ABB RobotStudio station: pyramid material handling.rsstn

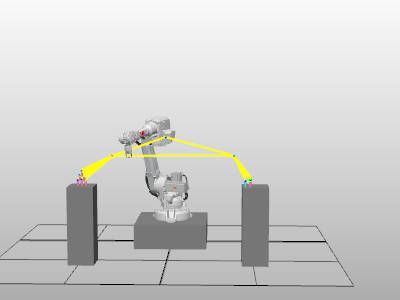
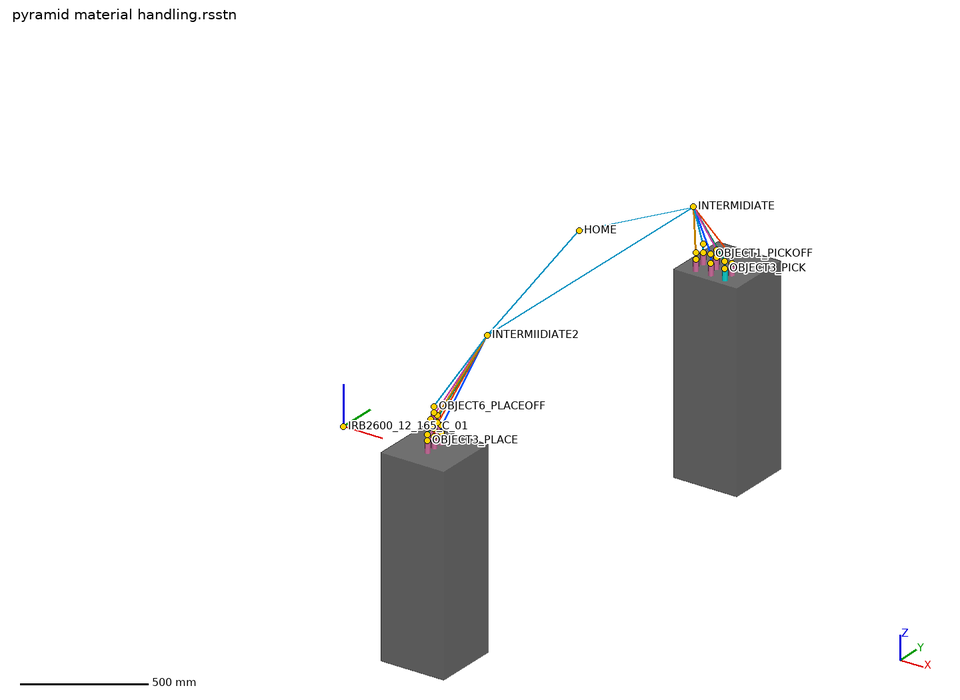
[picture v1: parts stored in the station drawn from their meshes, with robot base, taught points and paths (robot models come from the ABB library and are not in the file)]
Station Station (saved by RobotStudio 22.3.10141.1)
Controller Controller22, task T_ROB1: task frame (RAPID world) sits at (0, 0, 300) mm in the station
Controller Controller22
  mechanical unit ROB_1: IRB2600_12_165_C_01, 6 joints, base frame (0, 0, 0) mm
Layout (positions relative to the parent item):
  - concrete [part, from Libraries\concrete.rslib] at (-450, -450, 0) mm
  - IRB2600_12_165_C_01 [mechanism, from %ABB.RobotStudio.Models.IRB2600%\IRB2600_12_165_C_01.rslib] at (0, 0, 300) mm; joint values [-0.383, 0.3414, -0.2454, 0.1215, 1.4907, -1.8238] (rad or m)
  - SmartComponent_1 [smart component] at (1103.4, -433.44, 1358.47) mm, rotated rx -179.18 ry 6.95 rz -98.01 deg
      signals: DI attach
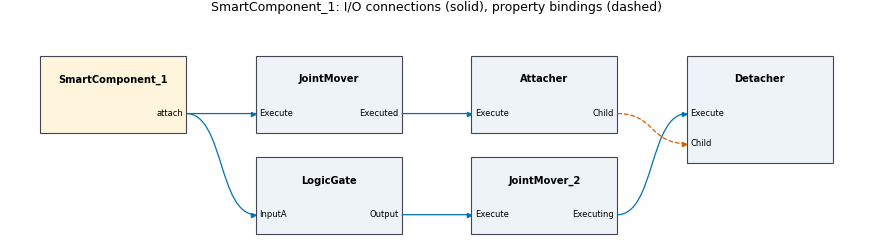
      connections:
        SmartComponent_1.attach -> JointMover.Execute
        JointMover.Executed -> Attacher.Execute
        SmartComponent_1.attach -> LogicGate.InputA
        LogicGate.Output -> JointMover_2.Execute
        JointMover_2.Executing -> Detacher.Execute
        Attacher.Child => Detacher.Child
    - Smart_Gripper_Servo_Fingers [mechanism, from Tools\ABB_Smart_Gripper_Servo_Fingers.rslib] at (0, 0, 0) mm; joint values [0.025] (rad or m)
    - JointMover [smart component, from Components\JointMover.rslib]
        properties: Mechanism=Smart_Gripper_Servo_Fingers; Relative=false; Duration=1; J1=0.023
    - JointMover_2 [smart component, from Components\JointMover.rslib]
        properties: Mechanism=Smart_Gripper_Servo_Fingers; Relative=false; Duration=1; J1=0.025
    - Attacher [smart component, from Components\Attacher.rslib]
        properties: Parent=Smart_Gripper_Servo_Fingers; Flange=0; Child=object_2; Mount=true; Offset=[0 0 0]; Orientation=[0 0 0]
    - LogicGate [smart component, from Components\LogicGate.rslib]
        properties: Operator=NOT; Delay=0
    - Detacher [smart component, from Components\Detacher.rslib]
        properties: Child=object_2; KeepPosition=true
  - table_1 [part] at (955.3, 870.39, 0) mm, size 300 x 300 x 900 mm
  - table_2 [part] at (955.3, -1114.68, 0) mm, size 300 x 300 x 900 mm
  - object [part] at (1175.36, 905.1, 900) mm, size 24 x 23.9 x 50 mm
  - object_2 [part] at (1105.3, 910.78, 900) mm, size 24 x 23.9 x 50 mm
  - object_3 [part] at (1035.28, 908.05, 900) mm, size 24 x 23.9 x 50 mm
  - object_4 [part] at (1171.86, 957.54, 900) mm, size 24 x 23.9 x 50 mm
  - object_5 [part] at (1089.6, 967.64, 900) mm, size 24 x 23.9 x 50 mm
  - object_6 [part] at (1025.27, 972.61, 900) mm, size 24 x 23.9 x 50 mm
  - object_7 [part] at (1105.3, -918.27, 900) mm, size 24 x 23.9 x 50 mm
  - object_8 [part] at (1105.3, -987.65, 951.01) mm, size 24 x 23.9 x 50 mm
  - object_9 [part] at (1105.3, -963.96, 900) mm, size 24 x 23.9 x 50 mm
  - object_10 [part] at (1105.3, -1009.85, 900) mm, size 24 x 23.9 x 50 mm
  - object_11 [part] at (1101.97, -962.11, 1002.3) mm, size 24 x 23.9 x 50 mm
  - object_12 [part] at (1104, -939.48, 950.56) mm, size 24 x 23.9 x 50 mm
Attachment: SmartComponent_1 is attached to IRB2600_12_165_C_01 / Link6
Station logic (signal -> signal, property => property):
  Controller22.attach -> SmartComponent_1.attach
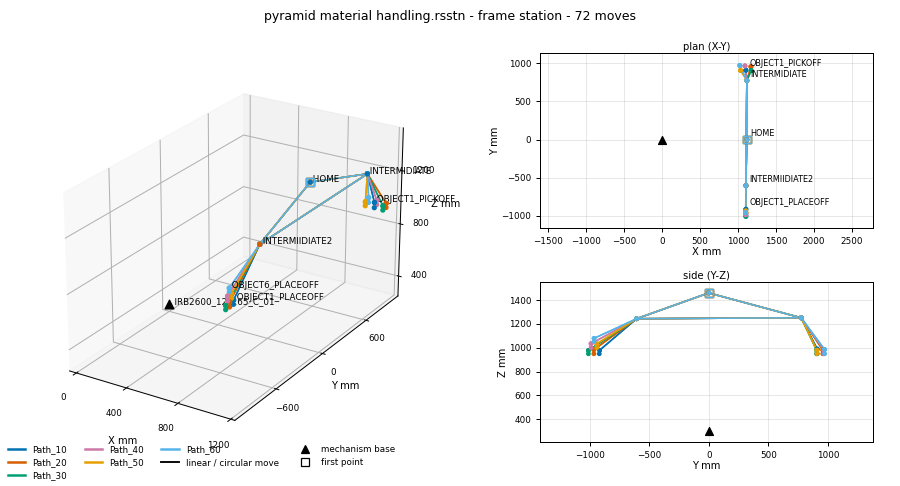
[picture p0: tool path of pyramid material handling.rsstn in frame station, 72 of 72 moves have a stored position in this frame; points joined in program order, loops and branches not executed]
Targets, tools, work objects and paths stored in the station, written as RAPID:
! task T_ROB1
MODULE CalibData
  PERS tooldata Servo:=[TRUE,[[0,0,114.2],[1,0,0,0]],[0.215,[8.7,12.3,49.2],[1,0,0,0],0.00021,0.00024,0.00009]];
ENDMODULE

! task T_ROB1
MODULE Module1
  CONST robtarget HOME:=[[1117.512260434,0,1160.4],[0.5,0,0.866025404,0],[-1,0,-1,0],[9E+09,9E+09,9E+09,9E+09,9E+09,9E+09]];
  CONST robtarget INTERMIDIATE:=[[1117.511971759,775.742463489,951.918308096],[0.499999999,-0.000000019,0.866025404,-0.000000013],[0,-1,0,0],[9E+09,9E+09,9E+09,9E+09,9E+09,9E+09]];
  CONST robtarget OBJECT1_PICK:=[[1105.303025435,910.780920196,650.000496725],[0.031021397,0.726247096,-0.685674321,-0.038125503],[0,0,-1,0],[9E+09,9E+09,9E+09,9E+09,9E+09,9E+09]];
  CONST robtarget OBJECT1_PICKOFF:=[[1105.303029888,910.780922429,689.758722238],[0.031021402,0.726247091,-0.685674327,-0.038125501],[0,0,-1,0],[9E+09,9E+09,9E+09,9E+09,9E+09,9E+09]];
  CONST robtarget INTERMIIDIATE2:=[[1105.30303417,-605.615476166,944.068794255],[0.031021378,0.726247007,-0.685674414,-0.038125531],[-1,-1,-2,0],[9E+09,9E+09,9E+09,9E+09,9E+09,9E+09]];
  CONST robtarget OBJECT1_PLACEOFF:=[[1105.303024526,-915.788819642,679.371711603],[0.031021384,0.726246988,-0.685674432,-0.038125586],[-1,-1,-2,0],[9E+09,9E+09,9E+09,9E+09,9E+09,9E+09]];
  CONST robtarget OBJECT1_PLACE:=[[1105.303040834,-918.273374791,650.000557068],[0.048952776,0.997947113,0.041056953,-0.004417227],[-1,-1,-3,0],[9E+09,9E+09,9E+09,9E+09,9E+09,9E+09]];
  CONST robtarget OBJECT2_PICKOFF:=[[1171.854966869,957.544914108,680.827668552],[0.048952841,0.997947109,0.041056966,-0.004417275],[0,-1,2,0],[9E+09,9E+09,9E+09,9E+09,9E+09,9E+09]];
  CONST robtarget OBJECT2_PICK:=[[1171.854963575,957.544912565,650.000541945],[0.048952828,0.997947111,0.041056939,-0.004417259],[0,-1,2,0],[9E+09,9E+09,9E+09,9E+09,9E+09,9E+09]];
  CONST robtarget OBJECT2_PLACE:=[[1105.303062744,-963.963465372,650.000529902],[0.032980269,-0.000000014,0.999456003,-0.000000058],[-1,0,-1,0],[9E+09,9E+09,9E+09,9E+09,9E+09,9E+09]];
  CONST robtarget OBJECT2_PLACEOFF:=[[1105.303062826,-963.963348224,684.023309799],[0.032980254,-0.000000025,0.999456003,-0.000000041],[-1,0,-1,0],[9E+09,9E+09,9E+09,9E+09,9E+09,9E+09]];
  CONST robtarget OBJECT3_PICK:=[[1175.361028607,905.095684377,650.00036776],[0.032980272,-0.000000022,0.999456003,0.000000007],[0,-1,0,0],[9E+09,9E+09,9E+09,9E+09,9E+09,9E+09]];
  CONST robtarget OBJECT3_PICKOFF:=[[1175.361033546,905.095684913,680.920223597],[0.032980305,-0.000000024,0.999456002,0.000000024],[0,-1,0,0],[9E+09,9E+09,9E+09,9E+09,9E+09,9E+09]];
  CONST robtarget OBJECT3_PLACE:=[[1105.303017361,-1009.850990253,650.000518886],[0.012165324,-0.000000073,0.999926,0.00000009],[-1,0,-1,0],[9E+09,9E+09,9E+09,9E+09,9E+09,9E+09]];
  CONST robtarget OBJECT3_PLACEOFF:=[[1105.303018098,-1009.850992621,677.758682693],[0.012165313,-0.000000049,0.999926,0.000000096],[-1,0,-1,0],[9E+09,9E+09,9E+09,9E+09,9E+09,9E+09]];
  CONST robtarget OBJECT4_PICK:=[[1092.960961058,967.413179097,650.000592066],[0.012159249,-0.00038074,0.999436296,-0.031290549],[0,-1,0,0],[9E+09,9E+09,9E+09,9E+09,9E+09,9E+09]];
  CONST robtarget OBJECT4_PICKOFF:=[[1092.960942706,967.413161677,681.87987598],[0.012159227,-0.000380743,0.999436295,-0.031290571],[0,-1,0,0],[9E+09,9E+09,9E+09,9E+09,9E+09,9E+09]];
  CONST robtarget OBJECT4_PLACE:=[[1105.303059247,-987.652451485,701.005559379],[0.01215924,-0.000380764,0.999436295,-0.03129058],[-1,-1,-1,0],[9E+09,9E+09,9E+09,9E+09,9E+09,9E+09]];
  CONST robtarget OBJECT4_PLACEOFF:=[[1105.303051029,-987.65244336,734.548047629],[0.01215925,-0.000380769,0.999436295,-0.031290587],[-1,-1,-1,0],[9E+09,9E+09,9E+09,9E+09,9E+09,9E+09]];
  CONST robtarget OBJECT5_PICK:=[[1035.27796955,908.054796965,650.000524579],[0.012159264,-0.000380741,0.999436295,-0.031290572],[0,-1,0,0],[9E+09,9E+09,9E+09,9E+09,9E+09,9E+09]];
  CONST robtarget OBJECT5_PICKOFF:=[[1035.277973445,908.054801244,679.543184231],[0.012159231,-0.000380712,0.999436294,-0.031290599],[0,-1,0,0],[9E+09,9E+09,9E+09,9E+09,9E+09,9E+09]];
  CONST robtarget OBJECT6_PICK:=[[1025.27201636,972.608074292,650.00053276],[0.012159217,-0.000380717,0.999436295,-0.031290601],[0,-1,0,0],[9E+09,9E+09,9E+09,9E+09,9E+09,9E+09]];
  CONST robtarget OBJECT6_PICKOFF:=[[1025.272009872,972.608069219,685.945409595],[0.012159225,-0.000380706,0.999436295,-0.031290591],[0,-1,0,0],[9E+09,9E+09,9E+09,9E+09,9E+09,9E+09]];
  CONST robtarget OBJECT5_PLACE:=[[1104.003999984,-939.476367792,700.564025373],[0.036344455,-0.000000046,0.999339322,0.000000022],[-1,0,-1,0],[9E+09,9E+09,9E+09,9E+09,9E+09,9E+09]];
  CONST robtarget OBJECT5_PLACEOFF:=[[1104.004008474,-939.47637643,733.669576361],[0.036344447,-0.000000033,0.999339322,0.000000026],[-1,0,-1,0],[9E+09,9E+09,9E+09,9E+09,9E+09,9E+09]];
  CONST robtarget OBJECT6_PLACE:=[[1101.97104085,-962.10978134,752.298904228],[0.036344493,0.000000006,0.999339321,0.000000002],[-1,0,-1,0],[9E+09,9E+09,9E+09,9E+09,9E+09,9E+09]];
  CONST robtarget OBJECT6_PLACEOFF:=[[1101.971036878,-962.109777758,779.422905783],[0.036344506,-0.000000004,0.99933932,-0.00000001],[-1,0,-1,0],[9E+09,9E+09,9E+09,9E+09,9E+09,9E+09]];
  PROC main()
  ENDPROC
  PROC Path_10()
    MoveL HOME,v1000,z100,Servo\WObj:=wobj0;
    MoveL INTERMIDIATE,v1000,z100,Servo\WObj:=wobj0;
    MoveL OBJECT1_PICKOFF,v1000,z100,Servo\WObj:=wobj0;
    MoveL OBJECT1_PICK,v1000,z100,Servo\WObj:=wobj0;
    WaitTime 1;
    SetDO attach,1;
    WaitTime 1;
    MoveL OBJECT1_PICKOFF,v1000,z100,Servo\WObj:=wobj0;
    MoveL INTERMIDIATE,v1000,z100,Servo\WObj:=wobj0;
    MoveL INTERMIIDIATE2,v1000,z100,Servo\WObj:=wobj0;
    MoveL OBJECT1_PLACEOFF,v1000,z100,Servo\WObj:=wobj0;
    MoveL OBJECT1_PLACE,v1000,z100,Servo\WObj:=wobj0;
    WaitTime 1;
    SetDO attach,0;
    WaitTime 1;
    MoveL OBJECT1_PLACEOFF,v1000,z100,Servo\WObj:=wobj0;
    MoveL INTERMIIDIATE2,v1000,z100,Servo\WObj:=wobj0;
    MoveL HOME,v1000,z100,Servo\WObj:=wobj0;
  ENDPROC
  PROC Path_20()
    MoveL HOME,v1000,z100,Servo\WObj:=wobj0;
    MoveL INTERMIDIATE,v1000,z100,Servo\WObj:=wobj0;
    MoveL OBJECT2_PICKOFF,v1000,z100,Servo\WObj:=wobj0;
    MoveL OBJECT2_PICK,v1000,z100,Servo\WObj:=wobj0;
    WaitTime 1;
    SetDO attach,1;
    WaitTime 1;
    MoveL OBJECT2_PICKOFF,v1000,z100,Servo\WObj:=wobj0;
    MoveL INTERMIDIATE,v1000,z100,Servo\WObj:=wobj0;
    MoveL INTERMIIDIATE2,v1000,z100,Servo\WObj:=wobj0;
    MoveL OBJECT2_PLACEOFF,v1000,z100,Servo\WObj:=wobj0;
    MoveL OBJECT2_PLACE,v1000,z100,Servo\WObj:=wobj0;
    WaitTime 1;
    SetDO attach,0;
    WaitTime 1;
    MoveL OBJECT2_PLACEOFF,v1000,z100,Servo\WObj:=wobj0;
    MoveL INTERMIIDIATE2,v1000,z100,Servo\WObj:=wobj0;
    MoveL HOME,v1000,z100,Servo\WObj:=wobj0;
  ENDPROC
  PROC Path_30()
    MoveL HOME,v1000,z100,Servo\WObj:=wobj0;
    MoveL INTERMIDIATE,v1000,z100,Servo\WObj:=wobj0;
    MoveL OBJECT3_PICKOFF,v1000,z100,Servo\WObj:=wobj0;
    MoveL OBJECT3_PICK,v1000,z100,Servo\WObj:=wobj0;
    WaitTime 1;
    SetDO attach,1;
    WaitTime 1;
    MoveL OBJECT3_PICKOFF,v1000,z100,Servo\WObj:=wobj0;
    MoveL INTERMIDIATE,v1000,z100,Servo\WObj:=wobj0;
    MoveL INTERMIIDIATE2,v1000,z100,Servo\WObj:=wobj0;
    MoveL OBJECT3_PLACEOFF,v1000,z100,Servo\WObj:=wobj0;
    MoveL OBJECT3_PLACE,v1000,z100,Servo\WObj:=wobj0;
    WaitTime 1;
    SetDO attach,0;
    WaitTime 1;
    MoveL OBJECT3_PLACEOFF,v1000,z100,Servo\WObj:=wobj0;
    MoveL INTERMIIDIATE2,v1000,z100,Servo\WObj:=wobj0;
    MoveL HOME,v1000,z100,Servo\WObj:=wobj0;
  ENDPROC
  PROC Path_40()
    MoveL HOME,v1000,z100,Servo\WObj:=wobj0;
    MoveL INTERMIDIATE,v1000,z100,Servo\WObj:=wobj0;
    MoveL OBJECT4_PICKOFF,v1000,z100,Servo\WObj:=wobj0;
    MoveL OBJECT4_PICK,v1000,z100,Servo\WObj:=wobj0;
    WaitTime 1;
    SetDO attach,1;
    WaitTime 1;
    MoveL OBJECT4_PICKOFF,v1000,z100,Servo\WObj:=wobj0;
    MoveL INTERMIDIATE,v1000,z100,Servo\WObj:=wobj0;
    MoveL INTERMIIDIATE2,v1000,z100,Servo\WObj:=wobj0;
    MoveL OBJECT4_PLACEOFF,v1000,z100,Servo\WObj:=wobj0;
    MoveL OBJECT4_PLACE,v1000,z100,Servo\WObj:=wobj0;
    WaitTime 1;
    SetDO attach,0;
    WaitTime 1;
    MoveL OBJECT4_PLACEOFF,v1000,z100,Servo\WObj:=wobj0;
    MoveL INTERMIIDIATE2,v1000,z100,Servo\WObj:=wobj0;
    MoveL HOME,v1000,z100,Servo\WObj:=wobj0;
  ENDPROC
  PROC Path_50()
    MoveL HOME,v1000,z100,Servo\WObj:=wobj0;
    MoveL INTERMIDIATE,v1000,z100,Servo\WObj:=wobj0;
    MoveL OBJECT5_PICKOFF,v1000,z100,Servo\WObj:=wobj0;
    MoveL OBJECT5_PICK,v1000,z100,Servo\WObj:=wobj0;
    WaitTime 1;
    SetDO attach,1;
    WaitTime 1;
    MoveL OBJECT5_PICKOFF,v1000,z100,Servo\WObj:=wobj0;
    MoveL INTERMIDIATE,v1000,z100,Servo\WObj:=wobj0;
    MoveL INTERMIIDIATE2,v1000,z100,Servo\WObj:=wobj0;
    MoveL OBJECT5_PLACEOFF,v1000,z100,Servo\WObj:=wobj0;
    MoveL OBJECT5_PLACE,v1000,z100,Servo\WObj:=wobj0;
    WaitTime 1;
    SetDO attach,0;
    WaitTime 1;
    MoveL OBJECT5_PLACEOFF,v1000,z100,Servo\WObj:=wobj0;
    MoveL INTERMIIDIATE2,v1000,z100,Servo\WObj:=wobj0;
    MoveL HOME,v1000,z100,Servo\WObj:=wobj0;
  ENDPROC
  PROC Path_60()
    MoveL HOME,v1000,z100,Servo\WObj:=wobj0;
    MoveL INTERMIDIATE,v1000,z100,Servo\WObj:=wobj0;
    MoveL OBJECT6_PICKOFF,v1000,z100,Servo\WObj:=wobj0;
    MoveL OBJECT6_PICK,v1000,z100,Servo\WObj:=wobj0;
    WaitTime 1;
    SetDO attach,1;
    WaitTime 1;
    MoveL OBJECT6_PICKOFF,v1000,z100,Servo\WObj:=wobj0;
    MoveL INTERMIDIATE,v1000,z100,Servo\WObj:=wobj0;
    MoveL INTERMIIDIATE2,v1000,z100,Servo\WObj:=wobj0;
    MoveL OBJECT6_PLACEOFF,v1000,z100,Servo\WObj:=wobj0;
    MoveL OBJECT6_PLACE,v1000,z100,Servo\WObj:=wobj0;
    WaitTime 1;
    SetDO attach,0;
    WaitTime 1;
    MoveL OBJECT6_PLACEOFF,v1000,z100,Servo\WObj:=wobj0;
    MoveL INTERMIIDIATE2,v1000,z100,Servo\WObj:=wobj0;
    MoveL HOME,v1000,z100,Servo\WObj:=wobj0;
  ENDPROC
  PROC Path_70()
    Path_10;
    Path_20;
    Path_30;
    Path_40;
    Path_50;
    Path_60;
  ENDPROC
ENDMODULE

